// TwinCAT 3 PLC project SampleProject
// libraries:
//   Tc2_Standard, * (Beckhoff Automation GmbH)
//   Tc2_System, 3.4.20.0 (Beckhoff Automation GmbH)
//   Base Interfaces,newest,System
// project tree:
//   / FB_Example.TcPOU, I_Example.TcPOU, PlcTask.TcTTO

CONFIGURATION SampleProject
    RESOURCE PLC ON TwinCAT3
        TASK PlcTask(INTERVAL := T#10ms, PRIORITY := 20);
        PROGRAM PRG_MAIN WITH PlcTask : PRG_MAIN;
    END_RESOURCE
END_CONFIGURATION

// ---- I_Example.TcPOU

// :Description: Example interface for TcKit parser validation.
INTERFACE I_Example


// :Description: Execute one cycle.
// :returns: TRUE when the operation completes
METHOD Execute : BOOL
VAR_INPUT
    bTrigger : BOOL;
END_VAR
END_METHOD


// :Description: Reset to idle state.
// :returns: TRUE on success
METHOD Reset : BOOL
END_METHOD


// :Description: Current status word.
PROPERTY Status : DWORD
GET
END_GET
END_PROPERTY

END_INTERFACE

// ---- FB_Example.TcPOU

// :Description: Example function block for TcKit parser validation.
// :param bEnable: Rising edge starts the operation
// :param nSetpoint: Target value in engineering units
FUNCTION_BLOCK FB_Example
VAR_INPUT
    bEnable    : BOOL;
    nSetpoint  : INT;
END_VAR
VAR_OUTPUT
    bDone      : BOOL;
    bError     : BOOL;
    nErrorId   : UDINT;
END_VAR
VAR
    eState     : E_ExampleState := E_ExampleState.Idle;
    nInternal  : INT;
END_VAR


CASE eState OF
    E_ExampleState.Idle:
        IF bEnable THEN
            eState := E_ExampleState.Running;
        END_IF

    E_ExampleState.Running:
        nInternal := nSetpoint;
        bDone := TRUE;
        eState := E_ExampleState.Idle;

    E_ExampleState.Error:
        bError := TRUE;
END_CASE


// :Description: Execute one cycle of the operation.
// :returns: TRUE when the operation completes successfully
METHOD Execute : BOOL
VAR_INPUT
    bTrigger : BOOL;
END_VAR

IF bTrigger THEN
    bDone := FALSE;
    bError := FALSE;
    nErrorId := 0;
    eState := E_ExampleState.Running;
END_IF

Execute := bDone;
END_METHOD


// :Description: Internal calculation used by the state machine.
METHOD CalculateInternal : INT
VAR_INPUT
    nFactor : INT;
END_VAR
VAR_OUTPUT
    bOverflow : BOOL;
END_VAR
VAR
    nScratch : DINT;
    bIntermediate : BOOL;
END_VAR
VAR_TEMP
    nTempResult : INT;
END_VAR
VAR CONSTANT
    nMaxValue : INT := 32767;
END_VAR

nScratch := nInternal * nFactor;
bOverflow := nScratch > nMaxValue;
nTempResult := INT_TO_INT(nScratch);
CalculateInternal := nTempResult;
END_METHOD


// :Description: Reset error state and outputs.
METHOD Reset : BOOL

bDone := FALSE;
bError := FALSE;
nErrorId := 0;
eState := E_ExampleState.Idle;
Reset := TRUE;
END_METHOD

ACTION LogState:

nInternal := nInternal;
END_ACTION


// :Description: Last error code, 0 when no error.
PROPERTY ErrorId : UDINT
GET

ErrorId := nErrorId;
END_GET
SET
VAR
    ErrorId : UDINT;
END_VAR

nErrorId := ErrorId;
END_SET
END_PROPERTY

END_FUNCTION_BLOCK
